TYPE st_EL2904Outputs :
STRUCT
	Output1 :BIT;
	Output2 :BIT;
	Output3 :BIT;
	Output4 :BIT;
	
END_STRUCT
END_TYPE

(* stored: Version 1.1.0.1, ProductVersion 3.1.4024.12
   DUT st_EL2904Outputs: Id {6b253499-d0b9-46ae-9478-ff5b3d7c6fd3} *)
